// TIA Portal V15.1 export
// export: Created 2020-06-12T07:35:54.7568359Z, ExportSetting None, DisplayName Totally Integrated Automation Portal, DisplayVersion V15.1, DisplayName TIA Portal Openness, DisplayVersion V15.1, DisplayName STEP 7 Professional, DisplayVersion V15.1, DisplayName STEP 7 Safety, DisplayVersion V15.1, DisplayName WinCC Advanced, DisplayVersion V15.1
FUNCTION "Desk_ctrl_act" : Void   // FC201, FBD
TITLE = Desk activation
{ S7_Optimized_Access := 'FALSE' }
// stored: AutoNumber false, SetENOAutomatically False
   VAR_TEMP
      _gt07_pulse_on : Bool;
      _gd01_pulse_on : Bool;
      _gd02_pulse_on : Bool;
      _gd03_pulse_on : Bool;
      _gd04_pulse_on : Bool;
      tDeactivate : Bool;
   END_VAR
BEGIN

REGION Network 1: desk +ES1GD01 activation
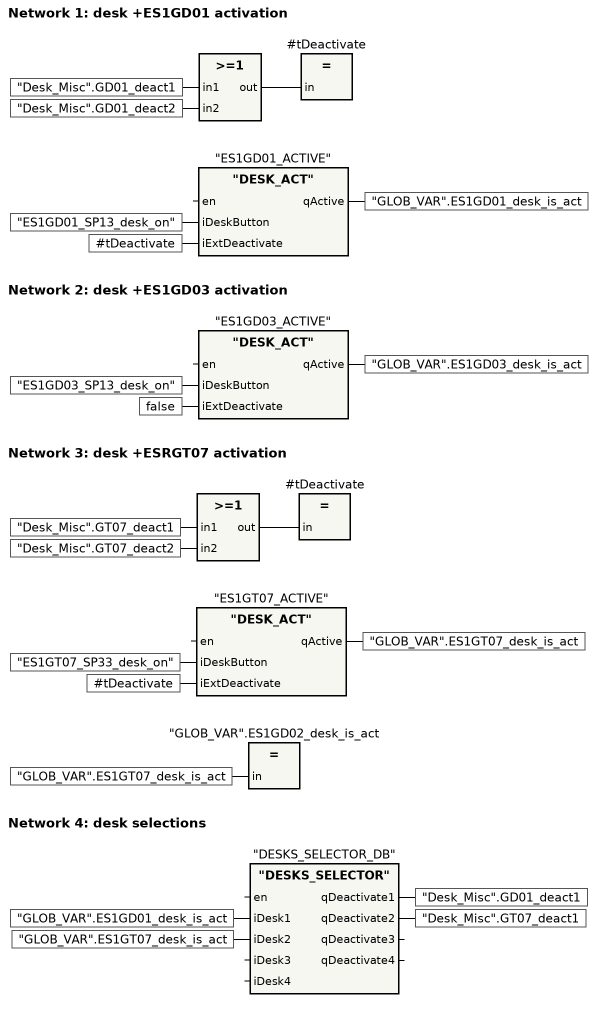
   #tDeactivate := "Desk_Misc".GD01_deact1 OR "Desk_Misc".GD01_deact2;
   "ES1GD01_ACTIVE"(iDeskButton := "ES1GD01_SP13_desk_on",   // "DESK_ACT"
                    iExtDeactivate := #tDeactivate,
                    qActive => "GLOB_VAR".ES1GD01_desk_is_act);
END_REGION

REGION Network 2: desk +ES1GD03 activation
   "ES1GD03_ACTIVE"(iDeskButton := "ES1GD03_SP13_desk_on",   // "DESK_ACT"
                    iExtDeactivate := false,
                    qActive => "GLOB_VAR".ES1GD03_desk_is_act);
END_REGION

REGION Network 3: desk +ESRGT07 activation
   #tDeactivate := "Desk_Misc".GT07_deact1 OR "Desk_Misc".GT07_deact2;
   "ES1GT07_ACTIVE"(iDeskButton := "ES1GT07_SP33_desk_on",   // "DESK_ACT"
                    iExtDeactivate := #tDeactivate,
                    qActive => "GLOB_VAR".ES1GT07_desk_is_act);
   "GLOB_VAR".ES1GD02_desk_is_act := "GLOB_VAR".ES1GT07_desk_is_act;
END_REGION

REGION Network 4: desk selections
   "DESKS_SELECTOR_DB"(iDesk1 := "GLOB_VAR".ES1GD01_desk_is_act,   // "DESKS_SELECTOR"
                       iDesk2 := "GLOB_VAR".ES1GT07_desk_is_act,
                       qDeactivate1 => "Desk_Misc".GD01_deact1,
                       qDeactivate2 => "Desk_Misc".GT07_deact1);
END_REGION
END_FUNCTION
